FUNCTION_BLOCK RejectWithMessageSyncHandler IMPLEMENTS I_SynchronousRpcHandler
VAR
END_VAR

METHOD Handle
VAR_INPUT
	Parameters : I_Deserializer;
	Response : I_SynchronousRpcResponse;
END_VAR
VAR
END_VAR
Response.RejectWithError('EXAMPLE_ERROR_CODE','This is the reject message');
END_METHOD

END_FUNCTION_BLOCK

(* stored: Version 1.1.0.1, ProductVersion 3.1.4026.13
   POU RejectWithMessageSyncHandler: Id {f7dd51c4-b7b4-0b91-25e7-17b220c50da2}, SpecialFunc None
   Method Handle: Id {cc098160-fa6a-0eca-2338-0c59c1006001} *)
